PROGRAM MAIN
VAR
	Profiler : PROFILER;
	ProfilerResult : PROFILERSTRUCT;

	fbCollision : FB_Collisions;
	fbRects : FB_initRects;
	bDone : BOOL := FALSE;
	
	collisionArray : ARRAY[0..29] OF BOOL;
	
	objectArray : ARRAY[ 0..maxObjects] OF stRect;
	
	bTriggerCppCode: BOOL := FALSE;
END_VAR

VAR CONSTANT
	maxObjects : INT := 300;
END_VAR


//Initialize Tines(circles) and Rectangles(objects/plants)
fbCollision.initCircles();
fbRects(rects := objectArray);

//Start timer
Profiler(START := TRUE, RESET := FALSE);
IF NOT bDone THEN
	bTriggerCppCode := TRUE; //Should trigger the Cpp code
END_IF

//Stop timer and publish results to view
Profiler(START := FALSE);
ProfilerResult := Profiler.DATA;

bDone := TRUE;

END_PROGRAM

(* stored: Version 1.1.0.1, ProductVersion 3.1.4026.8
   POU MAIN: Id {56430702-4f3b-488c-b8a0-85f48919f402}, SpecialFunc None *)
